INTERFACE I_VnRegister_Status

{attribute 'monitoring':='call'}
PROPERTY ReadDone : BOOL
GET
END_GET
END_PROPERTY

{attribute 'monitoring':='call'}
PROPERTY WriteDone : BOOL
GET
END_GET
END_PROPERTY

END_INTERFACE

(* stored: Version 1.1.0.1, ProductVersion 3.1.4024.12
   Itf I_VnRegister_Status: Id {4abec9b2-99ef-4920-b246-1713bdec0650}
   Property ReadDone: Id {a64668fc-38ec-496e-ad44-5b8d3187cae1}
   Get Get: Id {41bdfc70-33a8-46f8-9ae8-9b1ac717054a}
   Property WriteDone: Id {bc1db8c3-9212-4ae5-8894-d3f35f3f6930}
   Get Get: Id {978f1658-50be-4939-a2a1-d07157bebb1d} *)
